// TIA Portal V20 export
FUNCTION_BLOCK "AdjTop"   // FB520, FBD
{ S7_Optimized_Access := 'TRUE' }
// stored: AutoNumber false, MemoryReserve 100, SetENOAutomatically false
   VAR
      Var { ExternalAccessible := 'False'; ExternalVisible := 'False'; ExternalWritable := 'False'} : "TypeVar";
      Cmd { ExternalAccessible := 'False'; ExternalVisible := 'False'; ExternalWritable := 'False'} : "TypeCmd";
      Enc { ExternalAccessible := 'False'; ExternalVisible := 'False'; ExternalWritable := 'False'} : "SysCounterFast";
      Pos { ExternalAccessible := 'False'; ExternalVisible := 'False'; ExternalWritable := 'False'} : "SysPos";
      AdjSlow { ExternalAccessible := 'False'; ExternalVisible := 'False'; ExternalWritable := 'False'} : "SysMotor";
      AdjFast { ExternalAccessible := 'False'; ExternalVisible := 'False'; ExternalWritable := 'False'} : "SysLinMotC1150";
      TAutoOn { ExternalAccessible := 'False'; ExternalVisible := 'False'; ExternalWritable := 'False'} : TON_TIME;
      TAutoTarPosManOn { ExternalAccessible := 'False'; ExternalVisible := 'False'; ExternalWritable := 'False'} : TON_TIME;
      T { ExternalAccessible := 'False'; ExternalVisible := 'False'; ExternalWritable := 'False'} : Array[1..5] of IEC_TIMER;
      adjFastPnSlaveOff { ExternalAccessible := 'False'; ExternalVisible := 'False'; ExternalWritable := 'False'} : "SysPnSlaveDeactivate";
      tarOld { ExternalAccessible := 'False'; ExternalVisible := 'False'; ExternalWritable := 'False'} : DInt;
      autoTarPosMan { ExternalAccessible := 'False'; ExternalVisible := 'False'; ExternalWritable := 'False'} : Bool;
      setValueEnc { ExternalAccessible := 'False'; ExternalVisible := 'False'; ExternalWritable := 'False'} : Bool;
      autoRef { ExternalAccessible := 'False'; ExternalVisible := 'False'; ExternalWritable := 'False'} : Bool;
   END_VAR
   VAR_TEMP
      CtrlPc : Struct
         ackErr : Bool;
         manModeActive : Bool;
         manP : Bool;
         manM : Bool;
         manRefRun : Bool;
      END_STRUCT;
      CtrlLinMot : Struct
         Mode : Int;
         Target : Real;
         Speed : Real;
         Acc : Real;
         Dec : Real;
         Jerk : Real;
      END_STRUCT;
      refPosDiff : DInt;
      offsetNoStd : Real;
      refPosDiffCalib : DInt;
      modeCalib : Int;
      disMechanicToZero : Int;   // distance mechanic part top to zero [mm]
   END_VAR
   VAR_TEMP   // added for the SCL form of the ladder/FBD networks
      _w1 : Bool;
   END_VAR
BEGIN

REGION Network 1 (SCL): offset for no standard calibration
   (* 
   normally the distance from camera to board should be 550mm
   for special application the distance is different
   the distance can be changed in the goldeneye program
   if its different then 550mm a offset will be added
   *) 

   #offsetNoStd := 0.0;
   IF "ComRd".Data.Top.RefPosToBoard <> 550 THEN
       #offsetNoStd := (DINT_TO_REAL("ComRd".Data.Top.RefPosToBoard) - 550.0);
   END_IF;
END_REGION

REGION Network 2 (SCL): calibration value for offset
   (* 
   modus for calibartion
   camera must be referenced first
   mode 1 -->   the camera must be moved manually to position 550mm from board and
                 then press "Set Nullpoint"
   mode 2 -->   the camera must be moved to a other position and
                 then must be measured from the calibration tool to the camera and
                 this value must be putted in after pressing "Set Nullpoint"
   *)        
   #disMechanicToZero := 963;

   #modeCalib := 2;
   IF #modeCalib = 1 THEN
       #refPosDiffCalib := "ComRd".Data.Top.TargetPos;
   ELSIF #modeCalib = 2 THEN
       #refPosDiffCalib := (#disMechanicToZero * 10) - ("ComRd".Data.Top.CalibratePos + 5500);
   END_IF;
END_REGION

REGION Network 3 (SCL): calibration value from pc
   "ComSd".Data.Top.SetCalibratePosOk := FALSE;

   IF "ComRd".Data.Top.SetCalibratePos THEN

       IF "G".Cfg.adjTopActive THEN
           "Ref".adjTopCalOffset  := REAL_TO_DINT("Enc"."8BC1.T".act * 10.0) - #refPosDiffCalib;
       ELSIF "G".Cfg.adjTopActiveLinMot THEN
           "Ref".adjTopCalOffset  := REAL_TO_DINT("Enc"."8U1.T".act * 10.0) - #refPosDiffCalib;
       END_IF;

       "ComSd".Data.Top.SetCalibratePosOk := TRUE;
   END_IF;
END_REGION

REGION Network 4 (SCL): target position
   #Cmd.target := "G".Batch.thickness;
   IF ("G".Cfg.modeDimension = 3 OR "G".Cfg.modeDimension = 4) AND NOT "G".Batch.stdActive THEN
       #Cmd.target := "G".Batch.thicknessMeasure;
   END_IF;

   IF #autoTarPosMan THEN
       #Cmd.target := DINT_TO_REAL(("ComRd".Data.Top.TargetPos)) / 10.0;
   END_IF;

   "Ref".adjTopTar := #Cmd.target + (DINT_TO_REAL("Ref".adjTopCalOffset) / 10.0) + #offsetNoStd;
END_REGION

REGION Network 5 (SCL): data from pc
   IF NOT "G".errComPc THEN
       #CtrlPc.manModeActive := "ComRd".Data.Top.ManModeActive;
       #CtrlPc.manP := "ComRd".Data.Top.ManPlus;
       #CtrlPc.manM := "ComRd".Data.Top.ManMinus;
       #CtrlPc.manRefRun := "ComRd".Data.Top.ManRefRun;
   ELSE
       #CtrlPc.manModeActive := TRUE;
       #CtrlPc.manP := FALSE;
       #CtrlPc.manM := FALSE;
       #CtrlPc.manRefRun := FALSE;
   END_IF;

   #CtrlPc.ackErr := "G".ack;
END_REGION

REGION Network 6: off
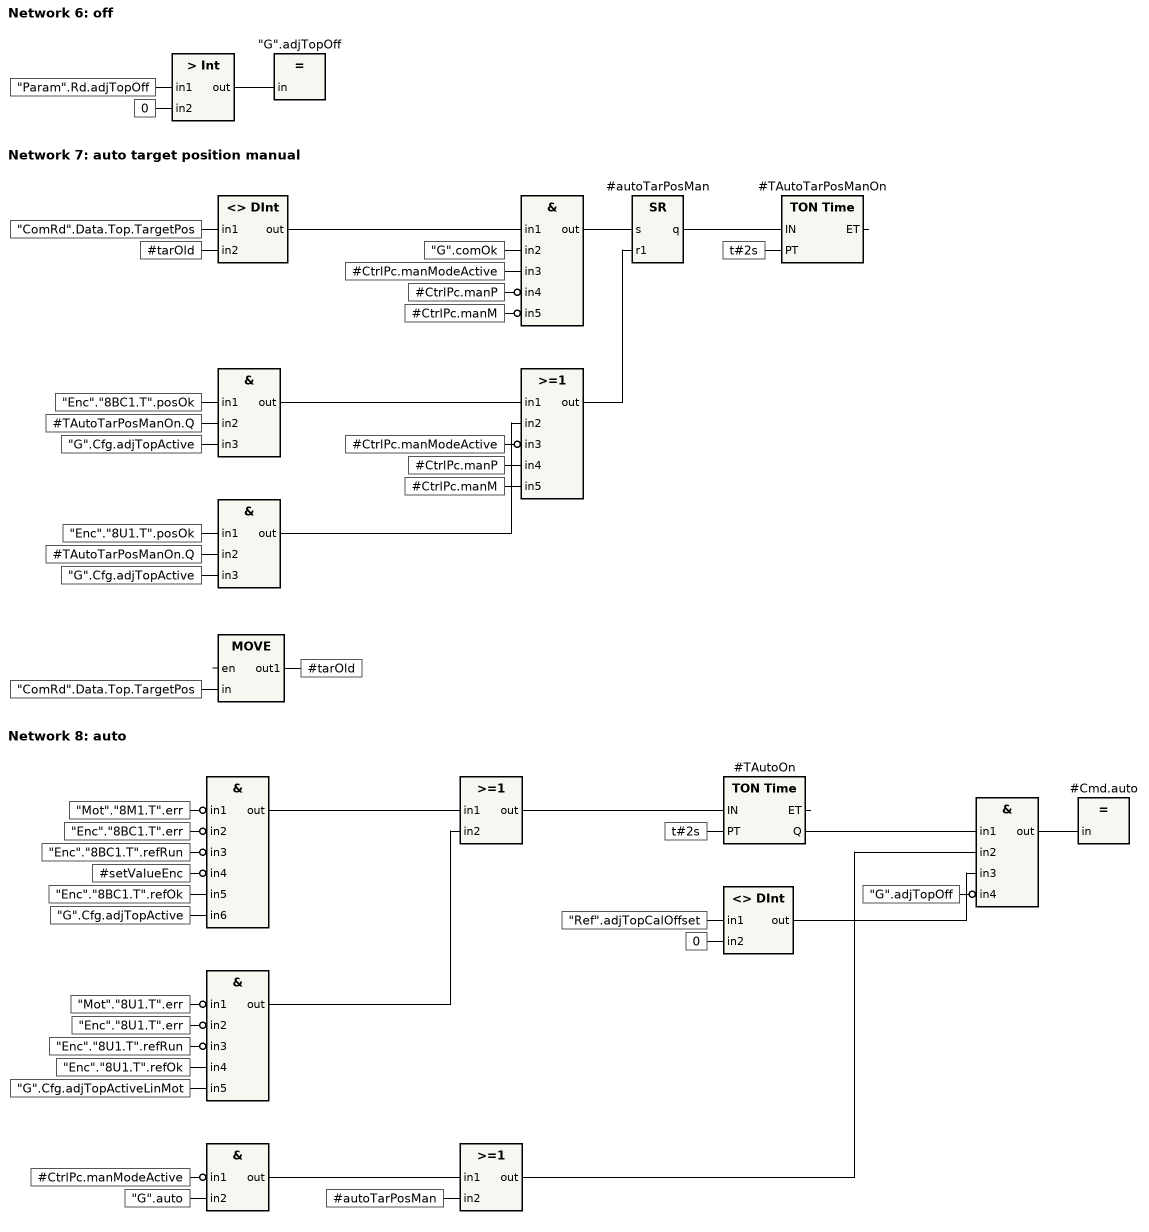
   "G".adjTopOff := "Param".Rd.adjTopOff > 0;
END_REGION

REGION Network 7: auto target position manual
   IF ("ComRd".Data.Top.TargetPos <> #tarOld) AND "G".comOk AND #CtrlPc.manModeActive AND NOT #CtrlPc.manP AND NOT #CtrlPc.manM THEN
       #autoTarPosMan := TRUE;   // SR flip-flop
   END_IF;
   IF ("Enc"."8BC1.T".posOk AND #TAutoTarPosManOn.Q AND "G".Cfg.adjTopActive) OR ("Enc"."8U1.T".posOk AND #TAutoTarPosManOn.Q AND "G".Cfg.adjTopActive) OR NOT #CtrlPc.manModeActive OR #CtrlPc.manP OR #CtrlPc.manM THEN
       #autoTarPosMan := FALSE;
   END_IF;
   #TAutoTarPosManOn(IN := #autoTarPosMan, PT := t#2s);   // TON
   #tarOld := "ComRd".Data.Top.TargetPos;
END_REGION

REGION Network 8: auto
   #TAutoOn(IN := (NOT "Mot"."8M1.T".err AND NOT "Enc"."8BC1.T".err AND NOT "Enc"."8BC1.T".refRun AND NOT #setValueEnc AND "Enc"."8BC1.T".refOk AND "G".Cfg.adjTopActive) OR (NOT "Mot"."8U1.T".err AND NOT "Enc"."8U1.T".err AND NOT "Enc"."8U1.T".refRun AND "Enc"."8U1.T".refOk AND "G".Cfg.adjTopActiveLinMot),   // TON
            PT := t#2s);
   #Cmd.auto := #TAutoOn.Q AND ((NOT #CtrlPc.manModeActive AND "G".auto) OR #autoTarPosMan) AND ("Ref".adjTopCalOffset <> 0) AND NOT "G".adjTopOff;
END_REGION

REGION Network 9: manual
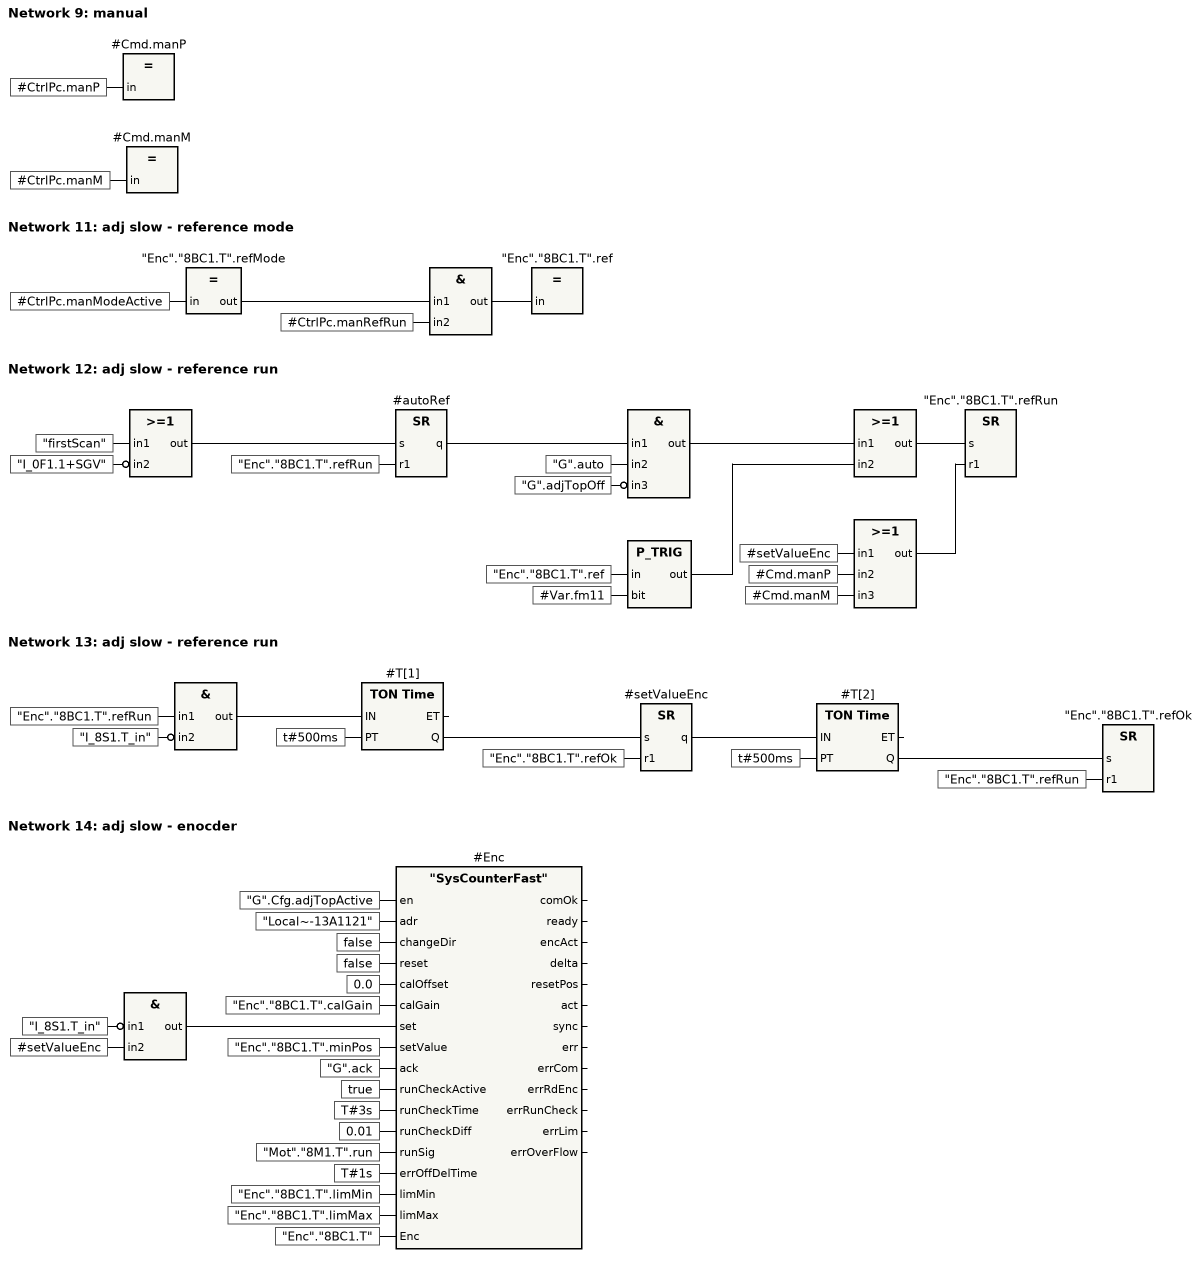
   #Cmd.manP := #CtrlPc.manP;
   #Cmd.manM := #CtrlPc.manM;
END_REGION

REGION Network 10 (SCL): adj slow - calibration value
   "Enc"."8BC1.T".calGain := -0.0275;

   "Enc"."8BC1.T".minPos := 10.0;
   "Enc"."8BC1.T".maxPos := 210.0;

   "Enc"."8BC1.T".limMin := "Enc"."8BC1.T".minPos - 5.0;
   "Enc"."8BC1.T".limMax := "Enc"."8BC1.T".maxPos + 5.0;

   "Enc"."8BC1.T".tarMinPos := "Enc"."8BC1.T".minPos + 0.0;
   "Enc"."8BC1.T".tarMaxPos := "Enc"."8BC1.T".maxPos - 0.0;
END_REGION

REGION Network 11: adj slow - reference mode
   "Enc"."8BC1.T".refMode := #CtrlPc.manModeActive;
   "Enc"."8BC1.T".ref := #CtrlPc.manModeActive AND #CtrlPc.manRefRun;
END_REGION

REGION Network 12: adj slow - reference run
   IF "firstScan" OR NOT "I_0F1.1+SGV" THEN
       #autoRef := TRUE;   // SR flip-flop
   END_IF;
   IF "Enc"."8BC1.T".refRun THEN #autoRef := FALSE; END_IF;
   #_w1 := "Enc"."8BC1.T".ref AND NOT #Var.fm11;   // rising edge
   #Var.fm11 := "Enc"."8BC1.T".ref;
   IF (#autoRef AND "G".auto AND NOT "G".adjTopOff) OR #_w1 THEN
       "Enc"."8BC1.T".refRun := TRUE;   // SR flip-flop
   END_IF;
   IF #setValueEnc OR #Cmd.manP OR #Cmd.manM THEN "Enc"."8BC1.T".refRun := FALSE; END_IF;
END_REGION

REGION Network 13: adj slow - reference run
   #T[1].TON(IN := "Enc"."8BC1.T".refRun AND NOT "I_8S1.T_in", PT := t#500ms);
   IF #T[1].Q THEN
       #setValueEnc := TRUE;   // SR flip-flop
   END_IF;
   IF "Enc"."8BC1.T".refOk THEN #setValueEnc := FALSE; END_IF;
   #T[2].TON(IN := #setValueEnc, PT := t#500ms);
   IF #T[2].Q THEN
       "Enc"."8BC1.T".refOk := TRUE;   // SR flip-flop
   END_IF;
   IF "Enc"."8BC1.T".refRun THEN "Enc"."8BC1.T".refOk := FALSE; END_IF;
END_REGION

REGION Network 14: adj slow - enocder
   IF "G".Cfg.adjTopActive THEN
       #Enc(adr := "Local~-13A1121",   // "SysCounterFast"
            changeDir := false,
            reset := false,
            calOffset := 0.0,
            calGain := "Enc"."8BC1.T".calGain,
            set := NOT "I_8S1.T_in" AND #setValueEnc,
            setValue := "Enc"."8BC1.T".minPos,
            ack := "G".ack,
            runCheckActive := true,
            runCheckTime := T#3s,
            runCheckDiff := 0.01,
            runSig := "Mot"."8M1.T".run,
            errOffDelTime := T#1s,
            limMin := "Enc"."8BC1.T".limMin,
            limMax := "Enc"."8BC1.T".limMax,
            Enc := "Enc"."8BC1.T");
   END_IF;
END_REGION

REGION Network 15: adj slow - pos
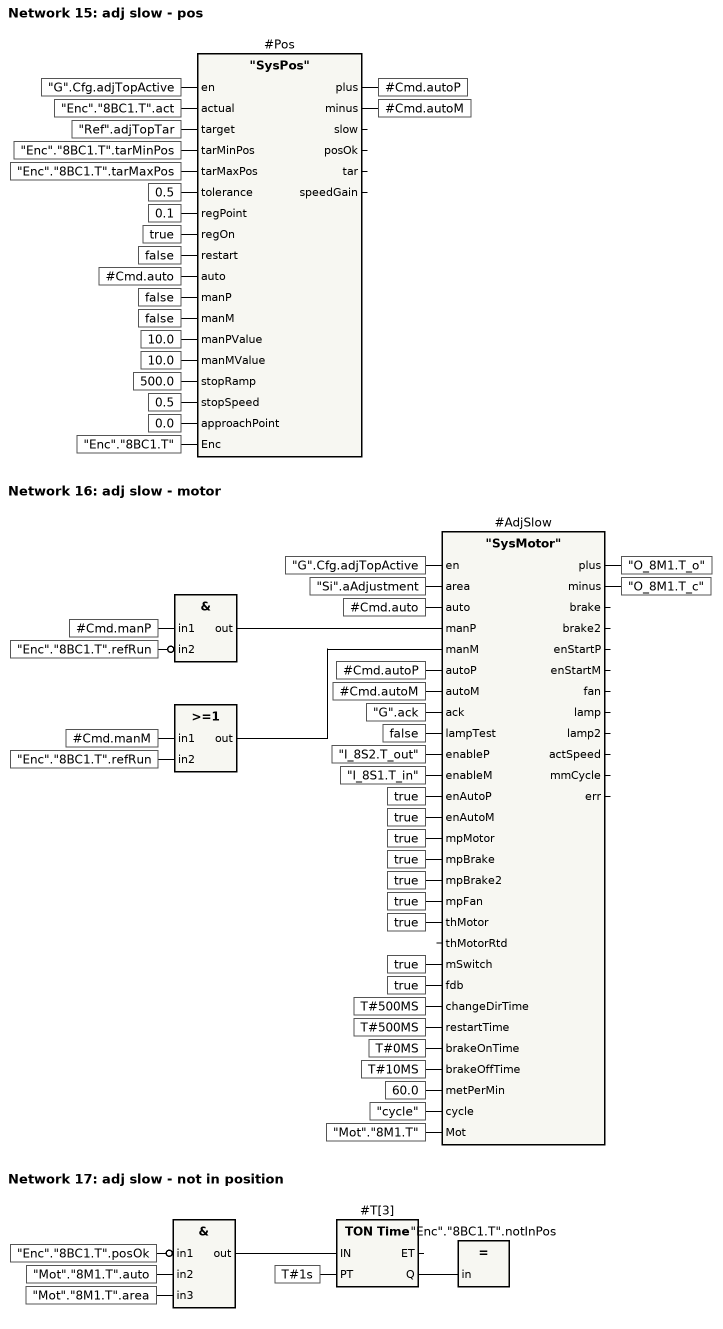
   IF "G".Cfg.adjTopActive THEN
       #Pos(actual := "Enc"."8BC1.T".act,   // "SysPos"
            target := "Ref".adjTopTar,
            tarMinPos := "Enc"."8BC1.T".tarMinPos,
            tarMaxPos := "Enc"."8BC1.T".tarMaxPos,
            tolerance := 0.5,
            regPoint := 0.1,
            regOn := true,
            restart := false,
            auto := #Cmd.auto,
            manP := false,
            manM := false,
            manPValue := 10.0,
            manMValue := 10.0,
            stopRamp := 500.0,
            stopSpeed := 0.5,
            approachPoint := 0.0,
            Enc := "Enc"."8BC1.T",
            plus => #Cmd.autoP,
            minus => #Cmd.autoM);
   END_IF;
END_REGION

REGION Network 16: adj slow - motor
   IF "G".Cfg.adjTopActive THEN
       #AdjSlow(area := "Si".aAdjustment,   // "SysMotor"
                auto := #Cmd.auto,
                manP := #Cmd.manP AND NOT "Enc"."8BC1.T".refRun,
                manM := #Cmd.manM OR "Enc"."8BC1.T".refRun,
                autoP := #Cmd.autoP,
                autoM := #Cmd.autoM,
                ack := "G".ack,
                lampTest := false,
                enableP := "I_8S2.T_out",
                enableM := "I_8S1.T_in",
                enAutoP := true,
                enAutoM := true,
                mpMotor := true,
                mpBrake := true,
                mpBrake2 := true,
                mpFan := true,
                thMotor := true,
                mSwitch := true,
                fdb := true,
                changeDirTime := T#500MS,
                restartTime := T#500MS,
                brakeOnTime := T#0MS,
                brakeOffTime := T#10MS,
                metPerMin := 60.0,
                cycle := "cycle",
                Mot := "Mot"."8M1.T",
                plus => "O_8M1.T_o",
                minus => "O_8M1.T_c");
   END_IF;
END_REGION

REGION Network 17: adj slow - not in position
   #T[3].TON(IN := NOT "Enc"."8BC1.T".posOk AND "Mot"."8M1.T".auto AND "Mot"."8M1.T".area, PT := T#1s);
   "Enc"."8BC1.T".notInPos := #T[3].Q;
END_REGION

REGION Network 18: adj slow - sensor monitoring
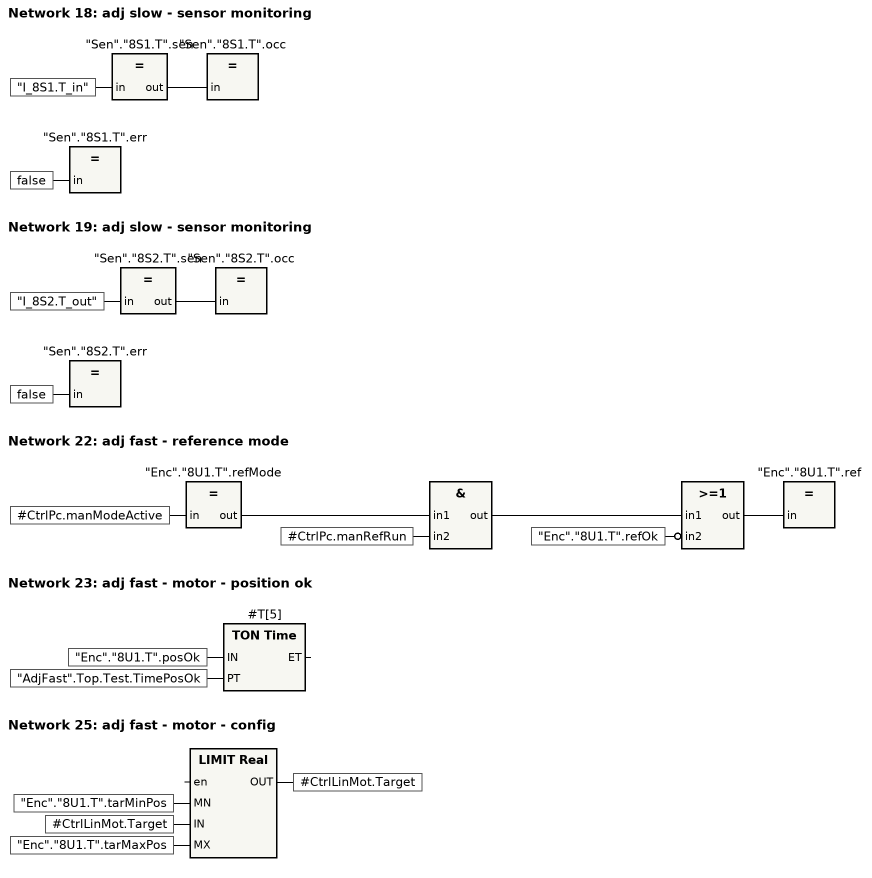
   "Sen"."8S1.T".sen := "I_8S1.T_in";
   "Sen"."8S1.T".occ := "I_8S1.T_in";
   "Sen"."8S1.T".err := false;
END_REGION

REGION Network 19: adj slow - sensor monitoring
   "Sen"."8S2.T".sen := "I_8S2.T_out";
   "Sen"."8S2.T".occ := "I_8S2.T_out";
   "Sen"."8S2.T".err := false;
END_REGION

REGION Network 21 (SCL): adj fast - calibration value
   "Enc"."8U1.T".calGain := 1.0;

   "Enc"."8U1.T".minPos := 5.0;
   "Enc"."8U1.T".maxPos := 155.0;

   "Enc"."8U1.T".limMin := "Enc"."8U1.T".minPos - 5.0;
   "Enc"."8U1.T".limMax := "Enc"."8U1.T".maxPos + 5.0;

   "Enc"."8U1.T".tarMinPos := "Enc"."8U1.T".minPos + 0.0;
   "Enc"."8U1.T".tarMaxPos := "Enc"."8U1.T".maxPos - 0.0;
END_REGION

REGION Network 22: adj fast - reference mode
   "Enc"."8U1.T".refMode := #CtrlPc.manModeActive;
   "Enc"."8U1.T".ref := (#CtrlPc.manModeActive AND #CtrlPc.manRefRun) OR NOT "Enc"."8U1.T".refOk;
END_REGION

REGION Network 23: adj fast - motor - position ok
   #T[5].TON(IN := "Enc"."8U1.T".posOk, PT := "AdjFast".Top.Test.TimePosOk);
END_REGION

REGION Network 24 (SCL): adj fast - motor - config

   //############################################################
   // min            5     mm
   // max          155     mm

   // speed        02      m/s
   // acc/dec      24      m/s2
   // jerk         450     m/s3

   // mode         BestehornVAJ
   //############################################################

   // only testmode for plc
   IF "AdjFast".Top.Test.ModeActive AND NOT #CtrlPc.manModeActive THEN
       IF "AdjFast".Top.Test.TarPos = "AdjFast".Top.Test.TarPos1 AND #T[5].Q THEN
           "AdjFast".Top.Test.TarPos := "AdjFast".Top.Test.TarPos2;
       ELSIF "AdjFast".Top.Test.TarPos = "AdjFast".Top.Test.TarPos2 AND #T[5].Q THEN
           "AdjFast".Top.Test.TarPos := "AdjFast".Top.Test.TarPos1;
       END_IF;
       "Ref".adjTopTar := "AdjFast".Top.Test.TarPos;
   END_IF;

   // active mode
   #CtrlLinMot.Mode := 3;
   #CtrlLinMot.Target := "Ref".adjTopTar;
   #CtrlLinMot.Speed := 2.0;
   #CtrlLinMot.Acc := 24.0;
   #CtrlLinMot.Dec := 0.0;
   #CtrlLinMot.Jerk := 450.0;

   // only testmode for plc
   IF "AdjFast".Top.Mode = 1 THEN
       #CtrlLinMot.Mode := 1;
       #CtrlLinMot.Target := "AdjFast".Top.VAI.Par1;
       #CtrlLinMot.Speed := "AdjFast".Top.VAI.Par2;
       #CtrlLinMot.Acc := "AdjFast".Top.VAI.Par3;
       #CtrlLinMot.Dec := "AdjFast".Top.VAI.Par4;
       #CtrlLinMot.Jerk := 0.0;
   ELSIF "AdjFast".Top.Mode = 2 THEN
       #CtrlLinMot.Mode := 2;
       #CtrlLinMot.Target := "AdjFast".Top.SinVA.Par1;
       #CtrlLinMot.Speed := "AdjFast".Top.SinVA.Par2;
       #CtrlLinMot.Acc := "AdjFast".Top.SinVA.Par3;
       #CtrlLinMot.Dec := 0.0;
       #CtrlLinMot.Jerk := 0.0;
   ELSIF "AdjFast".Top.Mode = 3 THEN
       #CtrlLinMot.Mode := 3;
       #CtrlLinMot.Target := "AdjFast".Top.BestehornVAJ.Par1;
       #CtrlLinMot.Speed := "AdjFast".Top.BestehornVAJ.Par2;
       #CtrlLinMot.Acc := "AdjFast".Top.BestehornVAJ.Par3;
       #CtrlLinMot.Dec := 0.0;
       #CtrlLinMot.Jerk := "AdjFast".Top.BestehornVAJ.Par4;
   END_IF;
END_REGION

REGION Network 25: adj fast - motor - config
   #CtrlLinMot.Target := LIMIT(MN := "Enc"."8U1.T".tarMinPos, IN := #CtrlLinMot.Target, MX := "Enc"."8U1.T".tarMaxPos);
END_REGION

REGION Network 26: adj fast - motor
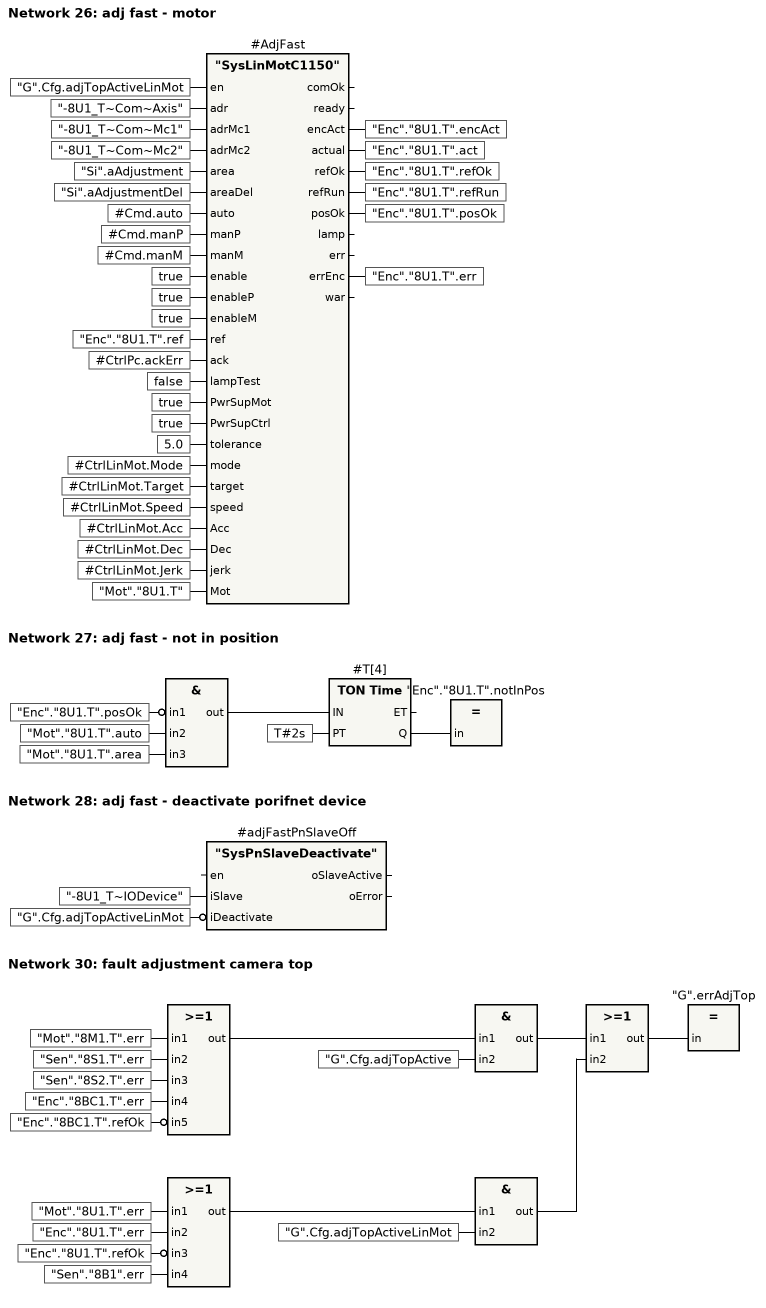
   IF "G".Cfg.adjTopActiveLinMot THEN
       #AdjFast(adr := "-8U1_T~Com~Axis",   // "SysLinMotC1150"
                adrMc1 := "-8U1_T~Com~Mc1",
                adrMc2 := "-8U1_T~Com~Mc2",
                area := "Si".aAdjustment,
                areaDel := "Si".aAdjustmentDel,
                auto := #Cmd.auto,
                manP := #Cmd.manP,
                manM := #Cmd.manM,
                enable := true,
                enableP := true,
                enableM := true,
                ref := "Enc"."8U1.T".ref,
                ack := #CtrlPc.ackErr,
                lampTest := false,
                PwrSupMot := true,
                PwrSupCtrl := true,
                tolerance := 5.0,
                mode := #CtrlLinMot.Mode,
                target := #CtrlLinMot.Target,
                speed := #CtrlLinMot.Speed,
                Acc := #CtrlLinMot.Acc,
                Dec := #CtrlLinMot.Dec,
                jerk := #CtrlLinMot.Jerk,
                Mot := "Mot"."8U1.T",
                encAct => "Enc"."8U1.T".encAct,
                actual => "Enc"."8U1.T".act,
                refOk => "Enc"."8U1.T".refOk,
                refRun => "Enc"."8U1.T".refRun,
                posOk => "Enc"."8U1.T".posOk,
                errEnc => "Enc"."8U1.T".err);
   END_IF;
END_REGION

REGION Network 27: adj fast - not in position
   #T[4].TON(IN := NOT "Enc"."8U1.T".posOk AND "Mot"."8U1.T".auto AND "Mot"."8U1.T".area, PT := T#2s);
   "Enc"."8U1.T".notInPos := #T[4].Q;
END_REGION

REGION Network 28: adj fast - deactivate porifnet device
   #adjFastPnSlaveOff(iSlave := "-8U1_T~IODevice", iDeactivate := NOT "G".Cfg.adjTopActiveLinMot);   // "SysPnSlaveDeactivate"
END_REGION

REGION Network 30: fault adjustment camera top
   "G".errAdjTop := (("Mot"."8M1.T".err OR "Sen"."8S1.T".err OR "Sen"."8S2.T".err OR "Enc"."8BC1.T".err OR NOT "Enc"."8BC1.T".refOk) AND "G".Cfg.adjTopActive) OR (("Mot"."8U1.T".err OR "Enc"."8U1.T".err OR NOT "Enc"."8U1.T".refOk OR "Sen"."8B1".err) AND "G".Cfg.adjTopActiveLinMot);
END_REGION

REGION Network 31 (SCL): data to pc
   IF "G".Cfg.adjTopActive THEN
       "Ref".adjTopAct := REAL_TO_DINT("Enc"."8BC1.T".act * 10.0) - "Ref".adjTopCalOffset - REAL_TO_DINT(#offsetNoStd * 10.0);
       "ComSd".Data.Top.ActualEncPos := REAL_TO_DINT("Enc"."8BC1.T".act * 10.0);
       "ComSd".Data.Top.ActualPos := "Ref".adjTopAct;
       "ComSd".Data.Top.LimitSwitchMin := "Sen"."8S1.T".sen;
       "ComSd".Data.Top.LimitSwitchMax := "Sen"."8S2.T".sen;
       "ComSd".Data.Top.Err := "Mot"."8M1.T".err;
       "ComSd".Data.Top.ErrEnc := "Enc"."8BC1.T".err;
       "ComSd".Data.Top.PosOk := "Enc"."8BC1.T".posOk;
       "ComSd".Data.Top.Plus := "Mot"."8M1.T".plus;
       "ComSd".Data.Top.Minus := "Mot"."8M1.T".minus;
       "ComSd".Data.Top.refRun := "Enc"."8BC1.T".refRun;
       "ComSd".Data.Top.refOk := "Enc"."8BC1.T".refOk;
   ELSIF  "G".Cfg.adjTopActiveLinMot THEN
       "Ref".adjTopAct := REAL_TO_DINT("Enc"."8U1.T".act * 10.0) - "Ref".adjTopCalOffset - REAL_TO_DINT(#offsetNoStd * 10.0);
       "ComSd".Data.Top.ActualEncPos := REAL_TO_DINT("Enc"."8U1.T".act * 10.0);
       "ComSd".Data.Top.ActualPos := "Ref".adjTopAct;
       "ComSd".Data.Top.LimitSwitchMin := TRUE;
       "ComSd".Data.Top.LimitSwitchMax := TRUE;
       "ComSd".Data.Top.Err := "Mot"."8U1.T".err;
       "ComSd".Data.Top.ErrEnc := "Enc"."8U1.T".err;
       "ComSd".Data.Top.PosOk := "Enc"."8U1.T".posOk;
       "ComSd".Data.Top.Plus := "Mot"."8U1.T".plus;
       "ComSd".Data.Top.Minus := "Mot"."8U1.T".minus;
       "ComSd".Data.Top.refRun := "Enc"."8U1.T".refRun;
       "ComSd".Data.Top.refOk := "Enc"."8U1.T".refOk;
   ELSE
       "ComSd".Data.Top.ActualEncPos := 0;
       "ComSd".Data.Top.ActualPos := 0;
       "ComSd".Data.Top.LimitSwitchMin := FALSE;
       "ComSd".Data.Top.LimitSwitchMax := FALSE;
       "ComSd".Data.Top.Err := FALSE;
       "ComSd".Data.Top.ErrEnc := FALSE;
       "ComSd".Data.Top.PosOk := True;
       "ComSd".Data.Top.Plus := FALSE;
       "ComSd".Data.Top.Minus := FALSE;
       "ComSd".Data.Top.refRun := FALSE;
       "ComSd".Data.Top.refOk := TRUE;
   END_IF;
END_REGION

REGION Network 32: current monitoring - auto
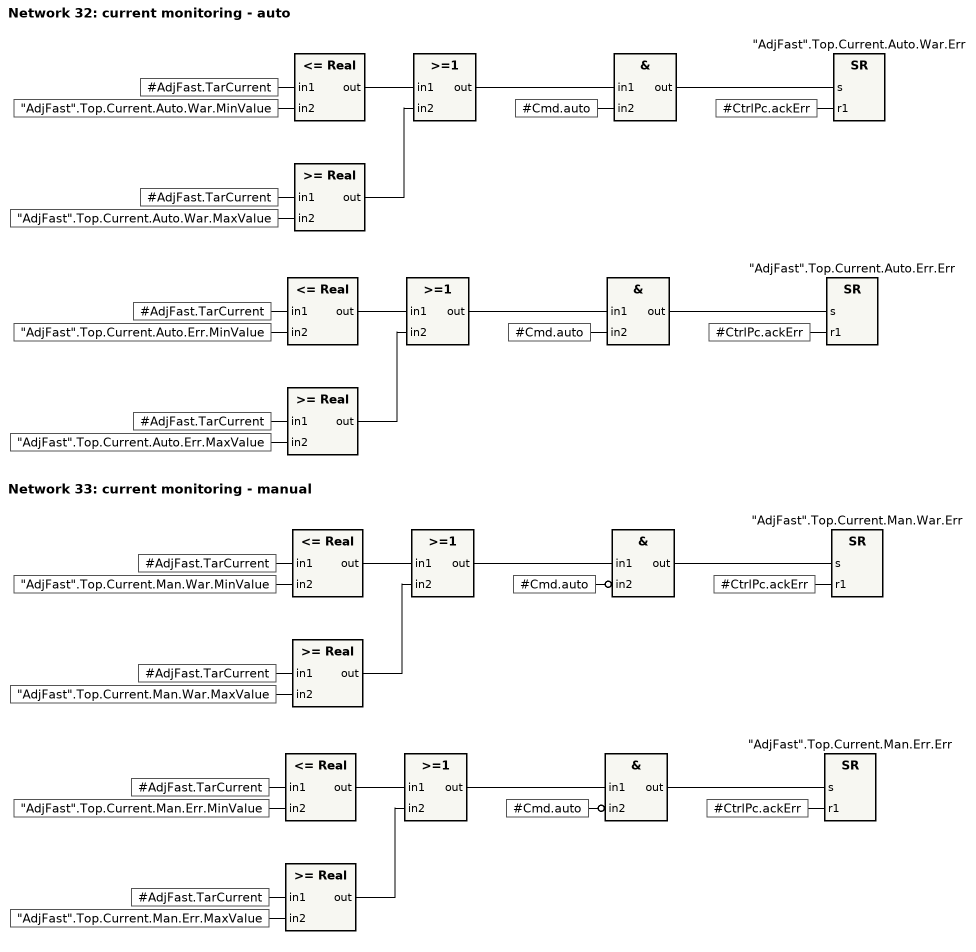
   IF ((#AdjFast.TarCurrent <= "AdjFast".Top.Current.Auto.War.MinValue) OR (#AdjFast.TarCurrent >= "AdjFast".Top.Current.Auto.War.MaxValue)) AND #Cmd.auto THEN
       "AdjFast".Top.Current.Auto.War.Err := TRUE;   // SR flip-flop
   END_IF;
   IF #CtrlPc.ackErr THEN "AdjFast".Top.Current.Auto.War.Err := FALSE; END_IF;
   IF ((#AdjFast.TarCurrent <= "AdjFast".Top.Current.Auto.Err.MinValue) OR (#AdjFast.TarCurrent >= "AdjFast".Top.Current.Auto.Err.MaxValue)) AND #Cmd.auto THEN
       "AdjFast".Top.Current.Auto.Err.Err := TRUE;   // SR flip-flop
   END_IF;
   IF #CtrlPc.ackErr THEN "AdjFast".Top.Current.Auto.Err.Err := FALSE; END_IF;
END_REGION

REGION Network 33: current monitoring - manual
   IF ((#AdjFast.TarCurrent <= "AdjFast".Top.Current.Man.War.MinValue) OR (#AdjFast.TarCurrent >= "AdjFast".Top.Current.Man.War.MaxValue)) AND NOT #Cmd.auto THEN
       "AdjFast".Top.Current.Man.War.Err := TRUE;   // SR flip-flop
   END_IF;
   IF #CtrlPc.ackErr THEN "AdjFast".Top.Current.Man.War.Err := FALSE; END_IF;
   IF ((#AdjFast.TarCurrent <= "AdjFast".Top.Current.Man.Err.MinValue) OR (#AdjFast.TarCurrent >= "AdjFast".Top.Current.Man.Err.MaxValue)) AND NOT #Cmd.auto THEN
       "AdjFast".Top.Current.Man.Err.Err := TRUE;   // SR flip-flop
   END_IF;
   IF #CtrlPc.ackErr THEN "AdjFast".Top.Current.Man.Err.Err := FALSE; END_IF;
END_REGION
END_FUNCTION_BLOCK
